// Mitsubishi GX Works2 project: BookEX6_54 Socket2   PLC: Q13UDV

// global labels: Global
VAR_GLOBAL
  bVar0 AT M5000 : BOOL;
  abArray0 AT M5010 : ARRAY [0..49] OF BOOL;
  sStr0 AT D5000 : STRING[199];
  sStr1 AT D5100 : STRING[199];
  sStr2 AT D5200 : STRING[199];
  sStr3 AT D5300 : STRING[199];
  sStr4 AT D5400 : STRING[199];
  sStr5 AT D5500 : STRING[199];
  sStr6 AT D5600 : STRING[199];
  sStr7 AT D5700 : STRING[199];
  sStr8 AT D5800 : STRING[199];
  sStr9 AT D5900 : STRING[199];
  iVar0 AT D4500 : INT;
  iVar1 AT D4501 : INT;
  iVar2 AT D4502 : INT;
  iVar3 AT D4503 : INT;
  iVar4 AT D4504 : INT;
  iVar5 AT D4505 : INT;
  iVar6 AT D4506 : INT;
  iVar7 AT D4507 : INT;
  iVar8 AT D4508 : INT;
  iVar9 AT D4509 : INT;
  dVar0 AT D4510 : DINT;
  dVar1 AT D4512 : DINT;
  dVar2 AT D4514 : DINT;
  dVar3 AT D4516 : DINT;
  dVar4 AT D4518 : DINT;
  dVar5 AT D4520 : DINT;
  dVar6 AT D4522 : DINT;
  dVar7 AT D4524 : DINT;
  dVar8 AT D4526 : DINT;
  dVar9 AT D4528 : DINT;
  wVar0 AT D4530 : WORD;
  wVar1 AT D4531 : WORD;
  wVar2 AT D4532 : WORD;
  wVar3 AT D4533 : WORD;
  wVar4 AT D4534 : WORD;
  wVar5 AT D4535 : WORD;
  wVar6 AT D4536 : WORD;
  wVar7 AT D4537 : WORD;
  wVar8 AT D4538 : WORD;
  wVar9 AT D4539 : WORD;
  dwVar0 AT D4540 : DWORD;
  dwVar1 AT D4542 : DWORD;
  dwVar2 AT D4544 : DWORD;
  dwVar3 AT D4546 : DWORD;
  dwVar4 AT D4548 : DWORD;
  dwVar5 AT D4550 : DWORD;
  dwVar6 AT D4552 : DWORD;
  dwVar7 AT D4554 : DWORD;
  dwVar8 AT D4556 : DWORD;
  dwVar9 AT D4558 : DWORD;
  fsVar0 AT D4560 : REAL;
  fsVar1 AT D4562 : REAL;
  fsVar2 AT D4564 : REAL;
  fsVar3 AT D4566 : REAL;
  fsVar4 AT D4568 : REAL;
  fsVar5 AT D4570 : REAL;
  fsVar6 AT D4572 : REAL;
  fsVar7 AT D4574 : REAL;
  fsVar8 AT D4576 : REAL;
  fsVar9 AT D4578 : REAL;
  fdVar0 AT D4580 : LREAL;
  tTime0 AT D4620 : TIME;
  tTime1 AT D4622 : TIME;
  tTime2 AT D4624 : TIME;
  tTime3 AT D4626 : TIME;
  tTime4 AT D4628 : TIME;
  tTime5 AT D4630 : TIME;
  tTime6 AT D4632 : TIME;
  tTime7 AT D4634 : TIME;
  tTime8 AT D4636 : TIME;
  tTime9 AT D4638 : TIME;
  tTime10 AT D4640 : TIME;
  bVar1 AT M5001 : BOOL;
  bVar2 AT M5002 : BOOL;
  bVar3 AT M5003 : BOOL;
  bVar4 AT M5004 : BOOL;
  bVar5 AT M5005 : BOOL;
  bVar6 AT M5006 : BOOL;
  bVar7 AT M5007 : BOOL;
  bVar8 AT M5008 : BOOL;
  bVar9 AT M5009 : BOOL;
  abArray1 AT M5060 : ARRAY [0..49] OF BOOL;
  abArray2 AT M5110 : ARRAY [0..49] OF BOOL;
  abArray3 AT M5160 : ARRAY [0..49] OF BOOL;
  abArray4 AT M5210 : ARRAY [0..49] OF BOOL;
  abArray5 AT M5260 : ARRAY [0..49] OF BOOL;
  abArray6 AT M5310 : ARRAY [0..49] OF BOOL;
  abArray7 AT M5360 : ARRAY [0..49] OF BOOL;
  abArray8 AT M5410 : ARRAY [0..49] OF BOOL;
  abArray9 AT M5460 : ARRAY [0..49] OF BOOL;
  fdVar1 AT D4584 : LREAL;
  fdVar2 AT D4588 : LREAL;
  fdVar3 AT D4592 : LREAL;
  fdVar4 AT D4596 : LREAL;
  fdVar5 AT D4600 : LREAL;
  fdVar6 AT D4604 : LREAL;
  fdVar7 AT D4608 : LREAL;
  fdVar8 AT D4612 : LREAL;
  fdVar9 AT D4616 : LREAL;
END_VAR

// global labels: QPLCSpecial
VAR_GLOBAL
  sbGetTime AT SM213 : BOOL;
  sbOn AT SM400 : BOOL;
  sbOff AT SM401 : BOOL;
  sbOn1Time AT SM402 : BOOL;
  sbOff1Time AT SM403 : BOOL;
  sb5ms AT SM409 : BOOL;
  sdSwitch AT SD200 : INT;
  sdTime03 AT SD212 : INT;
  sdTime04 AT SD213 : INT;
  sdTime02 AT SD211 : INT;
  sdTime01 AT SD210 : INT;
  sdScanTime1 AT SD521 : INT;
  sdScanTimeMin1 AT SD525 : INT;
  sdScanTimeMin AT SD524 : INT;
  sdScanTimeMax1 AT SD527 : INT;
  sdScanTimeMax AT SD526 : INT;
  sbErrInfo2 AT SM16 : BOOL;
  sbErrInfo AT SM5 : BOOL;
  sbSelfError AT SM1 : BOOL;
  sbDiagError AT SM0 : BOOL;
  sbResetErr AT SM50 : BOOL;
  sbSetTime AT SM210 : BOOL;
  sbFuse AT SM60 : BOOL;
  sbOpError AT SM56 : BOOL;
  sbPowerDown AT SM53 : BOOL;
  sbBatLow AT SM52 : BOOL;
  sbBatLowL AT SM51 : BOOL;
  sbSTOP AT SM203 : BOOL;
  sbPAUSE AT SM204 : BOOL;
  sbNsec AT SM414 : BOOL;
  sb1000ms AT SM413 : BOOL;
  sb500ms AT SM412 : BOOL;
  sbNms AT SM415 : BOOL;
  sbUserClk4 AT SM424 : BOOL;
  sbUserClk3 AT SM423 : BOOL;
  sbUserClk2 AT SM422 : BOOL;
  sbUserClk1 AT SM421 : BOOL;
  sbUserClk0 AT SM420 : BOOL;
  sdBatLowL AT SD51 : INT;
  sdPLCErrInfo AT SD4 : INT;
  sdPLCErrDate2 AT SD3 : INT;
  sdPLCErrDate1 AT SD2 : INT;
  sdPLCErrDate0 AT SD1 : INT;
  sdPLCErrCode AT SD0 : INT;
  sdFuse AT SD60 : INT;
  sdPowerDown AT SD53 : INT;
  sdBatLow AT SD52 : INT;
  sdCPUSts AT SD203 : INT;
  sdLed AT SD201 : INT;
  sdScanTime AT SD520 : INT;
  sdCntNsec AT SD414 : INT;
  sdCnt1sec AT SD412 : INT;
  sdCntScan AT SD420 : INT;
  sdCntNms AT SD415 : INT;
  sb100ms AT SM411 : BOOL;
  sb50ms AT SM410 : BOOL;
  sdSckOpenComp AT SD1282 : WORD;
  sdSckOpenReq AT SD1284 : WORD;
  sdSckDataRx AT SD1286 : WORD;
  sdSckConn AT SD1288 : WORD;
END_VAR

// global labels: Network
VAR_GLOBAL
  aSendData1 AT D100 : ARRAY [0..4] OF INT;
  aiTxData AT D4000 : ARRAY [0..99] OF INT;
  aiRxData AT D4100 : ARRAY [0..99] OF INT;
  iOpenOK AT D3900 : INT;
  iOpenERR AT D3901 : INT;
  iSendOK AT D3902 : INT;
  iSendERR AT D3903 : INT;
  iCloseOK AT D3906 : INT;
  iCloseERR AT D3907 : INT;
  iRecvOK AT D3904 : INT;
  iRecvERR AT D3905 : INT;
  aiTxData2 AT D4200 : ARRAY [0..99] OF INT;
  aiRxData2 AT D4300 : ARRAY [0..99] OF INT;
  iOpenOK2 AT D3908 : INT;
  iOpenERR2 AT D3909 : INT;
  iSendOK2 AT D3910 : INT;
  iSendERR2 AT D3911 : INT;
  iRecvOK2 AT D3912 : INT;
  iRecvERR2 AT D3913 : INT;
  iCloseOK2 AT D3914 : INT;
  iCloseERR2 AT D3915 : INT;
  iEOpenComp AT D3916 : INT;
  iEOpenReq AT D3917 : INT;
  iERecvFlag AT D3918 : INT;
  iOpenCode AT D3919 : INT;
  iSendCode AT D3920 : INT;
  iRecvCode AT D3921 : INT;
  iCloseCode AT D3922 : INT;
  iOpenCode2 AT D3923 : INT;
  iSendCode2 AT D3924 : INT;
  iRecvCode2 AT D3925 : INT;
  iCloseCode2 AT D3926 : INT;
  aRecvData1 AT D105 : ARRAY [0..4] OF INT;
  aSendData2 AT D110 : ARRAY [0..4] OF INT;
  aRecvData2 AT D115 : ARRAY [0..4] OF INT;
  aSendData3 AT D120 : ARRAY [0..4] OF INT;
  aRecvData3 AT D125 : ARRAY [0..4] OF INT;
  aRdata AT D140 : ARRAY [0..9] OF INT;
  aSLMPDataTx AT D150 : ARRAY [0..9] OF WORD;
  aSLMPDataRx AT D160 : ARRAY [0..9] OF WORD;
END_VAR
// user libraries (not included): HMI

PROGRAM Ex_READ
VAR
  Mov8INT_1 : Mov8INT;
  acRdCtrl : ARRAY [0..17] OF INT;
  abRdComp : ARRAY [0..1] OF BOOL;
  iCntRdOk : INT;
  iCntRdErr : INT;
END_VAR
(* structured ladder/FBD written out as ST: instructions are called as NAME(EN, inputs, outputs); _pN, _eN, _tN stand for wires *)
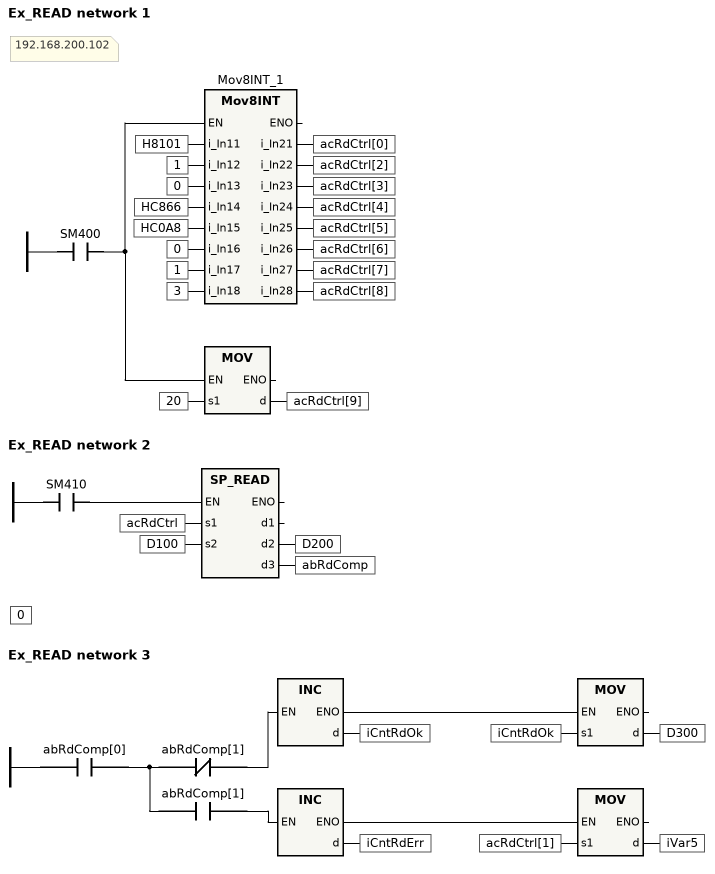
(* network 1 *)
(* 192.168.200.102 *)
Mov8INT_1(EN := SM400, i_In11 := H8101, i_In12 := 1, i_In13 := 0, i_In14 := HC866, i_In15 := HC0A8, i_In16 := 0, i_In17 := 1, i_In18 := 3, i_In21 => acRdCtrl[0], i_In22 => acRdCtrl[2], i_In23 => acRdCtrl[3], i_In24 => acRdCtrl[4], i_In25 => acRdCtrl[5], i_In26 => acRdCtrl[6], i_In27 => acRdCtrl[7], i_In28 => acRdCtrl[8]);
MOV(SM400, 20, acRdCtrl[9]);
(* network 2 *)
SP_READ(SM410, acRdCtrl, D100, _open, D200, abRdComp);
(* not connected to any output: 0 *)
(* network 3 *)
_e1 := INC(abRdComp[0] AND NOT abRdComp[1], iCntRdOk);
MOV(_e1, iCntRdOk, D300);
_e2 := INC(abRdComp[0] AND abRdComp[1], iCntRdErr);
MOV(_e2, acRdCtrl[1], iVar5);
END_PROGRAM

FUNCTION_BLOCK Word2Bit8
VAR_INPUT
  IN : WORD;
END_VAR
VAR_OUTPUT
  Bit0 : BOOL;
  Bit1 : BOOL;
  Bit2 : BOOL;
  Bit3 : BOOL;
  Bit4 : BOOL;
  Bit5 : BOOL;
  Bit6 : BOOL;
  Bit7 : BOOL;
END_VAR
 
Bit0 := WORD_TO_BOOL(IN AND 16#0001);
Bit1 := WORD_TO_BOOL(SHR(IN AND 16#0002 , 1));
Bit2 := WORD_TO_BOOL(SHR(IN AND 16#0004 , 2));
Bit3 := WORD_TO_BOOL(SHR(IN AND 16#0008 , 3));
Bit4 := WORD_TO_BOOL(SHR(IN AND 16#0010 , 4));
Bit5 := WORD_TO_BOOL(SHR(IN AND 16#0020 , 5));
Bit6 := WORD_TO_BOOL(SHR(IN AND 16#0040 , 6));
Bit7 := WORD_TO_BOOL(SHR(IN AND 16#0080 , 7));
END_FUNCTION_BLOCK

FUNCTION_BLOCK Word2Bit16
VAR_INPUT
  bEN : BOOL;
END_VAR
VAR_OUTPUT
  Bit0 : BOOL;
  Bit1 : BOOL;
  Bit2 : BOOL;
  Bit3 : BOOL;
  Bit4 : BOOL;
  Bit5 : BOOL;
  Bit6 : BOOL;
  Bit7 : BOOL;
  Bit8 : BOOL;
  Bit9 : BOOL;
  Bit10 : BOOL;
  Bit11 : BOOL;
  Bit12 : BOOL;
  Bit13 : BOOL;
  Bit14 : BOOL;
  Bit15 : BOOL;
END_VAR
VAR_INPUT
  InWord : WORD;
END_VAR
VAR_OUTPUT
  bENO : BOOL;
END_VAR
VAR
  InVal : WORD;
END_VAR
 
bENO := bEN;
InVal :=InWord;
Bit0 := (InVal AND 16#0001) = H0001;
Bit1 := (InVal AND 16#0002) = H0002;
Bit2 := (InVal AND 16#0004) = H0004;
Bit3 := (InVal AND 16#0008) = H0008;
Bit4 := (InVal AND 16#0010) = H0010;
Bit5 := (InVal AND 16#0020) = H0020;
Bit6 := (InVal AND 16#0040) = H0040;
Bit7 := (InVal AND 16#0080) = H0080;
Bit8 := (InVal AND 16#0100) = H0100;
Bit9 := (InVal AND 16#0200) = H0200;
Bit10 := (InVal AND 16#0400) = H0400;
Bit11 := (InVal AND 16#0800) = H0800;
Bit12 := (InVal AND 16#1000) = H1000;
Bit13 := (InVal AND 16#2000) = H2000;
Bit14 := (InVal AND 16#4000) = H4000;
Bit15 := (InVal AND 16#8000) = H8000;

(*
Bit0 := WORD_TO_BOOL(IN AND 16#0001);
Bit1 := WORD_TO_BOOL(SHR(IN AND 16#0002 , 1));
Bit2 := WORD_TO_BOOL(SHR(IN AND 16#0004 , 2));
Bit3 := WORD_TO_BOOL(SHR(IN AND 16#0008 , 3));
Bit4 := WORD_TO_BOOL(SHR(IN AND 16#0010 , 4));
Bit5 := WORD_TO_BOOL(SHR(IN AND 16#0020 , 5));
Bit6 := WORD_TO_BOOL(SHR(IN AND 16#0040 , 6));
Bit7 := WORD_TO_BOOL(SHR(IN AND 16#0080 , 7));
 
Bit8 := WORD_TO_BOOL(SHR(IN AND 16#0100 , 8));
Bit9 := WORD_TO_BOOL(SHR(IN AND 16#0200 , 9));
Bit10 := WORD_TO_BOOL(SHR(IN AND 16#0400 , 10));
Bit11 := WORD_TO_BOOL(SHR(IN AND 16#0800 , 11));
Bit12 := WORD_TO_BOOL(SHR(IN AND 16#1000 , 12));
Bit13 := WORD_TO_BOOL(SHR(IN AND 16#2000 , 13));
Bit14 := WORD_TO_BOOL(SHR(IN AND 16#4000 , 14));
Bit15 := WORD_TO_BOOL(SHR(IN AND 16#8000 , 15));
*)
END_FUNCTION_BLOCK

PROGRAM Ex_ECPRTCL
VAR
  bOpenReqC : BOOL;
  bOpenOkC : BOOL;
  bOpenErrC : BOOL;
  abOpenResC : ARRAY [0..1] OF BOOL;
  acOpenData : ARRAY [0..9] OF INT;
  bSendReqC : BOOL;
  bSendOkC : BOOL;
  bSendErrC : BOOL;
  abSendResC : ARRAY [0..1] OF BOOL;
  acSendDataC : ARRAY [0..1] OF INT;
  bRecvOkC : BOOL;
  bRecvErrC : BOOL;
  abRecvResC : ARRAY [0..1] OF BOOL;
  bCloseReq : BOOL;
  bCloseOkC : BOOL;
  bCloseErrC : BOOL;
  abCloseResC : ARRAY [0..1] OF BOOL;
  acCloseData : ARRAY [0..1] OF INT;
  CntSend1 : INT;
  CntSend2 : INT;
  CntRecv1 : INT;
  CntRecv2 : INT;
  Mov4INT_1 : Mov4INT;
  Mov8INT_1 : Mov8INT;
  acRdCtrl : ARRAY [0..9] OF INT;
  Mov4INT_2 : Mov4INT;
  bOpenReqE : BOOL;
  bOpenOkE : BOOL;
  bOpenErrE : BOOL;
  abOpenResE : ARRAY [0..1] OF BOOL;
  bSendErrE : BOOL;
  bSendOkE : BOOL;
  bSendReqE : BOOL;
  abSendResE : ARRAY [0..1] OF BOOL;
  abRecvResE : ARRAY [0..1] OF BOOL;
  bRecvErrE : BOOL;
  bRecvOkE : BOOL;
  abCloseResE : ARRAY [0..1] OF BOOL;
  bCloseErrE : BOOL;
  bCloseOkE : BOOL;
  acSendDataE : ARRAY [0..1] OF INT;
  acRecvDataC : ARRAY [0..1] OF INT;
  acRecvDataE : ARRAY [0..1] OF INT;
  Word2Bit8_1 : Word2Bit8;
  Word2Bit8_2 : Word2Bit8;
  Word2Bit8_3 : Word2Bit8;
  Word2Bit8_4 : Word2Bit8;
  Word2Bit8_5 : Word2Bit8;
  Word2Bit8_6 : Word2Bit8;
  ErrCodeSC : INT;
  ErrCodeSE : INT;
  Mov4INT_3 : Mov4INT;
  bChangeReqC : BOOL;
  Mov4INT_4 : Mov4INT;
  acRmodeData : ARRAY [0..3] OF INT;
  TON_1 : TON;
  CntRecvErr1 : INT;
  CntRecvErr2 : INT;
  TON_2 : TON;
  ErrCodeRC : INT;
  ErrCodeRE : INT;
  bModeReq : BOOL;
  acRdata : ARRAY [0..1] OF INT;
  bCmdReq : BOOL;
  abRes : ARRAY [0..1] OF BOOL;
  bOK : BOOL;
  bERR : BOOL;
  Mov8INT_2 : Mov8INT;
END_VAR
(* structured ladder/FBD written out as ST: instructions are called as NAME(EN, inputs, outputs); _pN, _eN, _tN stand for wires *)
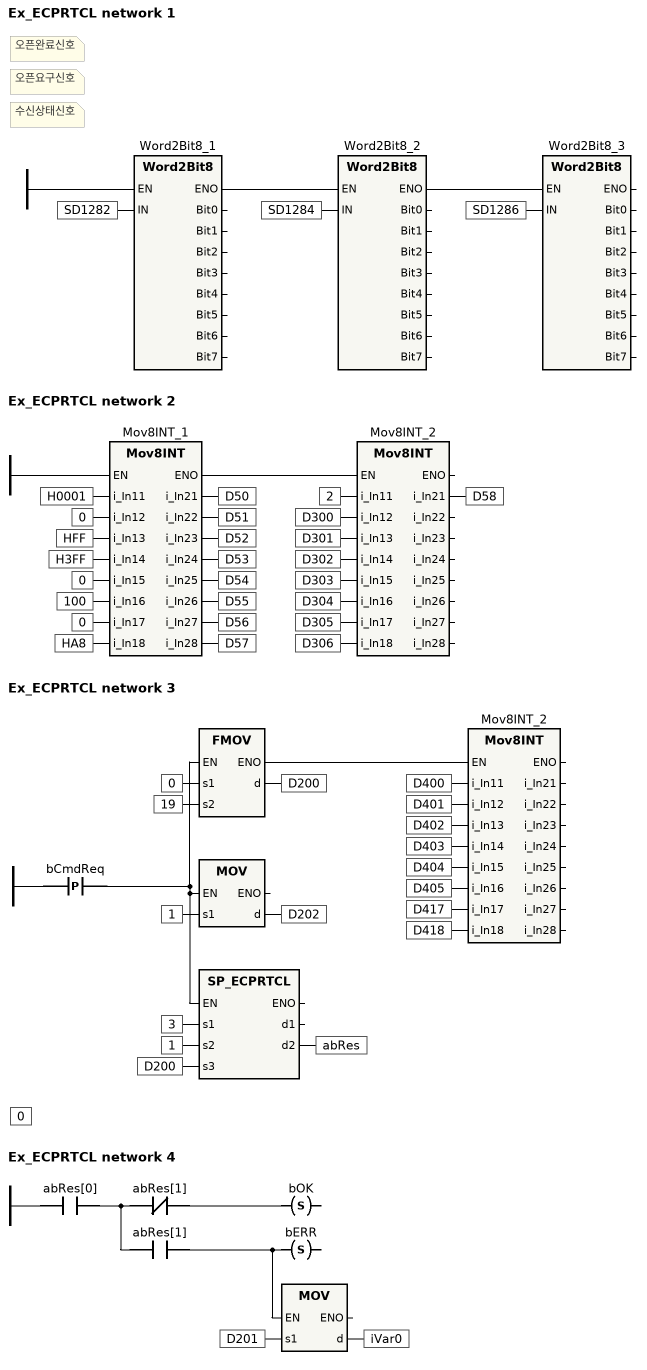
(* network 1 *)
(* 오픈완료신호 *)
(* 오픈요구신호 *)
(* 수신상태신호 *)
Word2Bit8_1(EN := TRUE, IN := SD1282);
Word2Bit8_2(EN := Word2Bit8_1.ENO, IN := SD1284);
Word2Bit8_3(EN := Word2Bit8_2.ENO, IN := SD1286);
(* network 2 *)
Mov8INT_1(EN := TRUE, i_In11 := H0001, i_In12 := 0, i_In13 := HFF, i_In14 := H3FF, i_In15 := 0, i_In16 := 100, i_In17 := 0, i_In18 := HA8, i_In21 => D50, i_In22 => D51, i_In23 => D52, i_In24 => D53, i_In25 => D54, i_In26 => D55, i_In27 => D56, i_In28 => D57);
Mov8INT_2(EN := Mov8INT_1.ENO, i_In11 := 2, i_In12 := D300, i_In13 := D301, i_In14 := D302, i_In15 := D303, i_In16 := D304, i_In17 := D305, i_In18 := D306, i_In21 => D58);
(* network 3 *)
_p1 := LDP(TRUE, bCmdReq);
_e2 := FMOV(_p1, 0, 19, D200);
Mov8INT_2(EN := _e2, i_In11 := D400, i_In12 := D401, i_In13 := D402, i_In14 := D403, i_In15 := D404, i_In16 := D405, i_In17 := D417, i_In18 := D418);
MOV(_p1, 1, D202);
SP_ECPRTCL(_p1, 3, 1, D200, _open, abRes);
(* not connected to any output: 0 *)
(* network 4 *)
SET(abRes[0] AND NOT abRes[1], bOK);
_p1 := abRes[0] AND abRes[1];
SET(_p1, bERR);
MOV(_p1, D201, iVar0);
END_PROGRAM

PROGRAM Ex_SLMPSND
VAR
  bSendReq : BOOL;
  Mov8WORD_1 : Mov8WORD;
  abSLMPRes : ARRAY [0..1] OF BOOL;
  acSLMPData : ARRAY [0..18] OF WORD;
  Mov8WORD_2 : Mov8WORD;
  Mov4WORD_1 : Mov4WORD;
  Mov8WORD_3 : Mov8WORD;
  Word2Bit16_1 : Word2Bit16;
  Word2Bit16_2 : Word2Bit16;
  Word2Bit16_3 : Word2Bit16;
  Word2Bit16_4 : Word2Bit16;
  abOpenResC : ARRAY [0..1] OF BOOL;
  abOpenResE : ARRAY [0..1] OF BOOL;
  acOpenData : ARRAY [0..9] OF INT;
  bOpenReqC : BOOL;
  bOpenOkC : BOOL;
END_VAR
(* structured ladder/FBD written out as ST: instructions are called as NAME(EN, inputs, outputs); _pN, _eN, _tN stand for wires *)
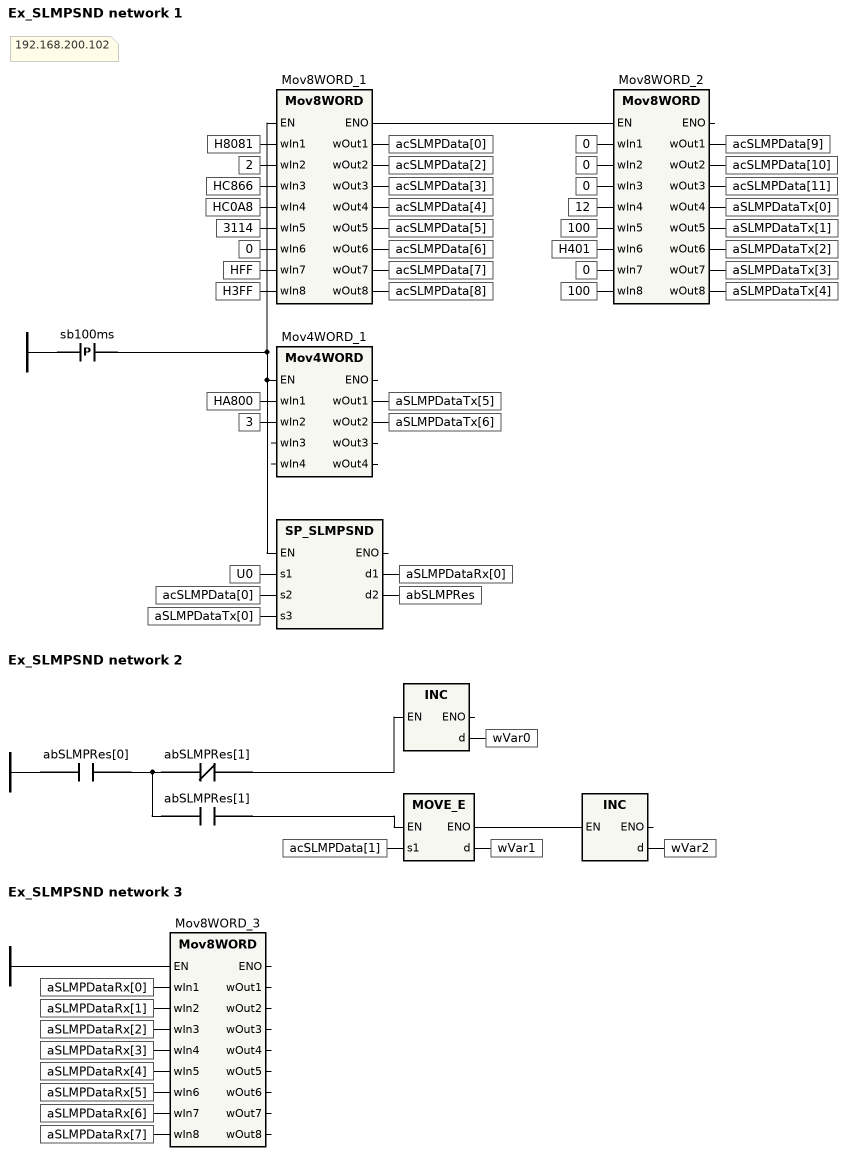
(* network 1 *)
(* 192.168.200.102 *)
_p1 := LDP(TRUE, sb100ms);
Mov8WORD_1(EN := _p1, wIn1 := H8081, wIn2 := 2, wIn3 := HC866, wIn4 := HC0A8, wIn5 := 3114, wIn6 := 0, wIn7 := HFF, wIn8 := H3FF, wOut1 => acSLMPData[0], wOut2 => acSLMPData[2], wOut3 => acSLMPData[3], wOut4 => acSLMPData[4], wOut5 => acSLMPData[5], wOut6 => acSLMPData[6], wOut7 => acSLMPData[7], wOut8 => acSLMPData[8]);
Mov8WORD_2(EN := Mov8WORD_1.ENO, wIn1 := 0, wIn2 := 0, wIn3 := 0, wIn4 := 12, wIn5 := 100, wIn6 := H401, wIn7 := 0, wIn8 := 100, wOut1 => acSLMPData[9], wOut2 => acSLMPData[10], wOut3 => acSLMPData[11], wOut4 => aSLMPDataTx[0], wOut5 => aSLMPDataTx[1], wOut6 => aSLMPDataTx[2], wOut7 => aSLMPDataTx[3], wOut8 => aSLMPDataTx[4]);
Mov4WORD_1(EN := _p1, wIn1 := HA800, wIn2 := 3, wOut1 => aSLMPDataTx[5], wOut2 => aSLMPDataTx[6]);
SP_SLMPSND(_p1, U0, acSLMPData[0], aSLMPDataTx[0], aSLMPDataRx[0], abSLMPRes);
(* network 2 *)
INC(abSLMPRes[0] AND NOT abSLMPRes[1], wVar0);
_e1 := MOVE_E(abSLMPRes[0] AND abSLMPRes[1], acSLMPData[1], wVar1);
INC(_e1, wVar2);
(* network 3 *)
Mov8WORD_3(EN := TRUE, wIn1 := aSLMPDataRx[0], wIn2 := aSLMPDataRx[1], wIn3 := aSLMPDataRx[2], wIn4 := aSLMPDataRx[3], wIn5 := aSLMPDataRx[4], wIn6 := aSLMPDataRx[5], wIn7 := aSLMPDataRx[6], wIn8 := aSLMPDataRx[7]);
END_PROGRAM

FUNCTION_BLOCK slmpDeviceRead
VAR_INPUT
  bEN : BOOL;
  dw_IPAddr : DWORD;
  i_SubCommand : INT;
  i_DeviceCode : INT;
  d_DeviceNo : DINT;
  i_DevicePoints : INT;
  i_Channel : INT;
  i_TargetPortNo : INT;
END_VAR
VAR_OUTPUT
  bENO : BOOL;
  b_OK : BOOL;
  b_ERR : BOOL;
  i_ErrCode : INT;
END_VAR
VAR
  aControlData : ARRAY [0..18] OF INT;
  aRequestData : ARRAY [0..7] OF INT;
  aResponesData : ARRAY [0..999] OF INT;
  abComp : ARRAY [0..1] OF BOOL;
  bErr1 : BOOL;
  bErr2 : BOOL;
  NoPoint : INT;
  TempDeviceCode : INT;
  bTmpErr : BOOL;
  bInputCheck : BOOL;
  bExecute : BOOL;
  bCheckEnd : BOOL;
END_VAR
VAR CONSTANT
  cRequestModuleIO : INT := H3FF;
  cResendCountMax : INT;
  cMonitorTime : INT := 1;
END_VAR
VAR
  dwTmp : DWORD;
END_VAR
VAR_OUTPUT
  i_ReadData : INT;
  i_ResendCount : INT;
  i_ErrTime : ARRAY [0..3] OF INT;
  dw_ErrIP : DWORD;
END_VAR
;
IF LDP(TRUE, bEN) AND NOT bENO THEN (*FB의 시작*)
	bENO 				:= TRUE;
	bInputCheck 	:= TRUE;
	b_OK 				:= FALSE;
	b_ERR 				:= FALSE;
	i_ErrCode 		:= 0;
	bTmpErr 			:= FALSE;
END_IF;

IF NOT bEN THEN (*FB의 종료*)
	b_OK 				:= FALSE;
	b_ERR 				:= FALSE;
	i_ErrCode 		:= 0;
 	bTmpErr 			:= FALSE;
	bENO 				:= FALSE;
	bInputCheck 	:= FALSE;
	bCheckEnd 	:= FALSE;
	bExecute 			:= FALSE;
END_IF;

IF LDP(TRUE, bInputCheck) THEN
	IF i_SubCommand < 0 OR i_SubCommand > 1 										THEN i_ErrCode := 11; END_IF;
	IF i_DeviceCode < 0 OR i_DeviceCode > WORD_TO_INT(HFF) 	THEN i_ErrCode := 12; END_IF;
	IF d_DeviceNo < 0 OR d_DeviceNo > DWORD_TO_DINT(HFFFFFF) 	THEN i_ErrCode := 13; END_IF;
	IF i_DevicePoints < 1 OR i_DevicePoints > 960 									THEN i_ErrCode := 14; END_IF;
	IF i_Channel < 1 OR i_Channel > 9 																THEN i_ErrCode := 15; END_IF;
	IF i_TargetPortNo = 0 OR i_TargetPortNo = HFFFF 							THEN i_ErrCode := 16; END_IF;
	IF i_ErrCode <> 0 THEN 		
		bTmpErr := TRUE;
	END_IF;	  
	bCheckEnd := bTmpErr = 0;
END_IF;			
		
IF LDP(TRUE, bCheckEnd) THEN
	FMOV(TRUE, 0, 19, aControlData[0]);		
	aControlData[0] 	:= H8081;
	aControlData[2] 	:= i_Channel;
	aControlData[3] 	:= DWORD_TO_INT(dw_IPAddr AND H0000FFFF);
	aControlData[4] 	:= DWORD_TO_INT(SHR(dw_IPAddr,16) AND H0000FFFF);
	aControlData[5] 	:= i_TargetPortNo;	
	aControlData[6] 	:= 0;	
	aControlData[7] 	:= HFF;	
	aControlData[8] 	:= cRequestModuleIO;	
	aControlData[9] 	:= 0;	
	aControlData[10] 	:= cResendCountMax;
	aControlData[11] 	:= cMonitorTime;

	aRequestData[0] := 12;
	aRequestData[1] := 2;
	aRequestData[2] := H401;
	aRequestData[3] := i_SubCommand;
	dwTmp := DINT_TO_DWORD( d_DeviceNo);
	aRequestData[4] := DWORD_TO_INT(dwTmp AND H0000FFFF);
	aRequestData[5] := DWORD_TO_INT(SHR(dwTmp,16) AND H0000FFFF);
	IF i_SubCommand = 0 THEN 
		NoPoint := i_DevicePoints; 
	ELSIF i_SubCommand = 1 THEN 
		NoPoint := i_DevicePoints+3; 
		NoPoint := i_DevicePoints / 4; 
	END_IF;
	TempDeviceCode := i_DeviceCode;
	SFL(TRUE, 8, TempDeviceCode);
	WOR(TRUE, TempDeviceCode, aRequestData[5], aRequestData[5]);
	aRequestData[6] := NoPoint;
	bExecute := TRUE;
END_IF;
			
SP_SLMPSND( bExecute, "U0", aControlData[0], aRequestData[0], aResponesData[0], abComp);  (*상승에지에서 실행*)
IF abComp[0] THEN	(*실행 완료 *)
	i_ErrCode 			:= aControlData[1];
	i_ResendCount 	:= aControlData[10];
	BMOV(TRUE, aControlData[13], 4, i_ErrTime[0]); 
	dw_ErrIP := INT_TO_DWORD(aControlData[17]) OR SHL(INT_TO_DWORD( aControlData[18]),16);
	bExecute 				:= FALSE;
	IF abComp[1] THEN
		bErr2 					:= TRUE;		(* 이상완료*)
	ELSE								(* 정상완료*)
		IF aResponesData[1] = 0 THEN
			b_OK 			:=TRUE;
		 	BMOV( TRUE, aResponesData[2], NoPoint, i_ReadData );
		ELSE
			i_ErrCode 	:= aResponesData[1];		(*에러코드*)
			bErr1 				:= TRUE; 
		END_IF;
	END_IF;
END_IF;

IF bTmpErr OR bErr1 OR bErr2 THEN
 	b_ERR 		:= TRUE;
 	bErr1 			:= FALSE;
  	bErr2 			:= FALSE;
END_IF;
END_FUNCTION_BLOCK

PROGRAM Ex_OtherUDV
VAR
  Mov8INT_1 : Mov8INT;
  Mov8INT_2 : Mov8INT;
END_VAR
(* structured ladder/FBD written out as ST: instructions are called as NAME(EN, inputs, outputs); _pN, _eN, _tN stand for wires *)
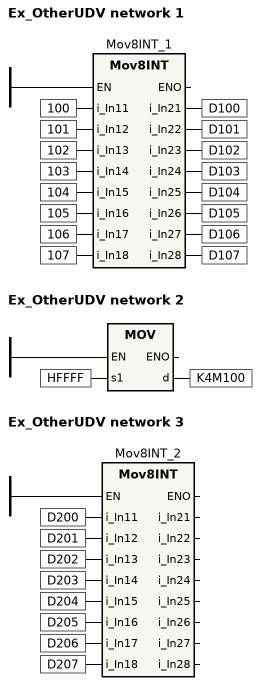
(* network 1 *)
Mov8INT_1(EN := TRUE, i_In11 := 100, i_In12 := 101, i_In13 := 102, i_In14 := 103, i_In15 := 104, i_In16 := 105, i_In17 := 106, i_In18 := 107, i_In21 => D100, i_In22 => D101, i_In23 => D102, i_In24 => D103, i_In25 => D104, i_In26 => D105, i_In27 => D106, i_In28 => D107);
(* network 2 *)
MOV(TRUE, HFFFF, K4M100);
(* network 3 *)
Mov8INT_2(EN := TRUE, i_In11 := D200, i_In12 := D201, i_In13 := D202, i_In14 := D203, i_In15 := D204, i_In16 := D205, i_In17 := D206, i_In18 := D207);
END_PROGRAM

PROGRAM Ex_DeviceRead
VAR
  slmpDeviceRead_1 : slmpDeviceRead;
  bRun : BOOL;
  bOK : BOOL;
  bERR : BOOL;
  ErrCode : INT;
  bSetErr : BOOL;
  bExeReq : BOOL;
  ResendCount : INT;
  ErrTime : ARRAY [0..3] OF INT;
  ErrIP : DWORD;
  Mov4INT_1 : Mov4INT;
  Mov4INT_2 : Mov4INT;
END_VAR
(* structured ladder/FBD written out as ST: instructions are called as NAME(EN, inputs, outputs); _pN, _eN, _tN stand for wires *)
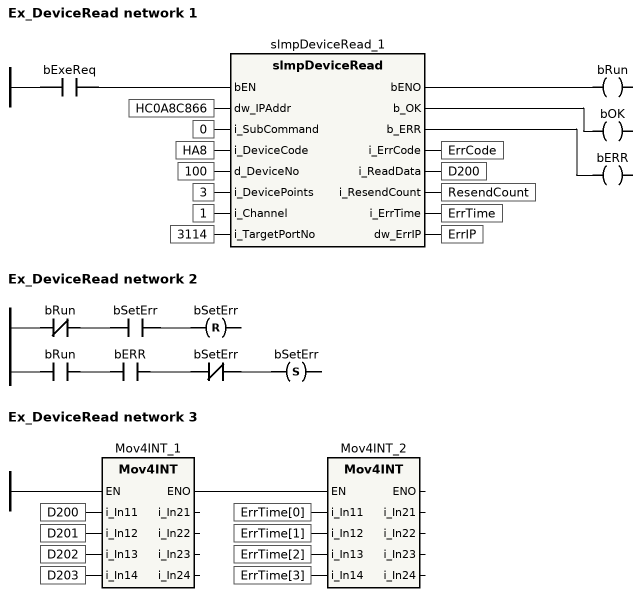
(* network 1 *)
slmpDeviceRead_1(bEN := bExeReq, dw_IPAddr := HC0A8C866, i_SubCommand := 0, i_DeviceCode := HA8, d_DeviceNo := 100, i_DevicePoints := 3, i_Channel := 1, i_TargetPortNo := 3114, i_ErrCode => ErrCode, i_ReadData => D200, i_ResendCount => ResendCount, i_ErrTime => ErrTime, dw_ErrIP => ErrIP);
bRun := slmpDeviceRead_1.bENO;
bOK := slmpDeviceRead_1.b_OK;
bERR := slmpDeviceRead_1.b_ERR;
(* network 2 *)
RST(NOT bRun AND bSetErr, bSetErr);
SET(bRun AND bERR AND NOT bSetErr, bSetErr);
(* network 3 *)
Mov4INT_1(EN := TRUE, i_In11 := D200, i_In12 := D201, i_In13 := D202, i_In14 := D203);
Mov4INT_2(EN := Mov4INT_1.ENO, i_In11 := ErrTime[0], i_In12 := ErrTime[1], i_In13 := ErrTime[2], i_In14 := ErrTime[3]);
END_PROGRAM

FUNCTION_BLOCK slmpDeviceWrite
VAR_INPUT
  bEN : BOOL;
  dw_IPAddr : DWORD;
  i_SubCommand : INT;
  i_DeviceCode : INT;
  d_DeviceNo : DINT;
  i_DevicePoints : INT;
  i_Channel : INT;
  i_TargetPortNo : INT;
END_VAR
VAR_OUTPUT
  bENO : BOOL;
  b_OK : BOOL;
  b_ERR : BOOL;
  i_ErrCode : INT;
END_VAR
VAR
  aControlData : ARRAY [0..18] OF INT;
  aRequestData : ARRAY [0..999] OF INT;
  aResponesData : ARRAY [0..6] OF INT;
  abComp : ARRAY [0..1] OF BOOL;
  NoWritePoint : INT;
  TempDeviceCode : INT;
  bTmpErr : BOOL;
  bInputCheck : BOOL;
  bExecute : BOOL;
  bCheckEnd : BOOL;
END_VAR
VAR CONSTANT
  cRequestModuleIO : INT := H3FF;
  cResendCountMax : INT;
  cMonitorTime : INT := 1;
END_VAR
VAR
  dwTmp : DWORD;
END_VAR
VAR_INPUT
  i_WriteData : INT;
END_VAR
VAR
  NoWriteLength : INT;
END_VAR
VAR_OUTPUT
  i_ResendCount : INT;
  i_ErrTime : ARRAY [0..3] OF INT;
  dw_ErrIP : DWORD;
END_VAR
VAR
  bErr1 : BOOL;
  bErr2 : BOOL;
END_VAR
;
IF LDP(TRUE, bEN) AND NOT bENO THEN (*FB의 시작*)
	bENO 				:= TRUE;
	bInputCheck 	:= TRUE;
	b_OK 				:= FALSE;
	b_ERR 				:= FALSE;
	i_ErrCode 		:= 0;
	bTmpErr 			:= FALSE;
END_IF;

IF NOT bEN THEN (*FB의 종료*)
	b_OK 				:= FALSE;
	b_ERR 				:= FALSE;
	i_ErrCode 		:= 0;
 	bTmpErr 			:= FALSE;
	bENO 				:= FALSE;
	bInputCheck 	:= FALSE;
	bCheckEnd 	:= FALSE;
	bExecute 			:= FALSE;
END_IF;

IF LDP(TRUE, bInputCheck) THEN
	IF i_SubCommand < 0 OR i_SubCommand > 1 										THEN i_ErrCode := 11; END_IF;
	IF i_DeviceCode < 0 OR i_DeviceCode > WORD_TO_INT(HFF) 	THEN i_ErrCode := 12; END_IF;
	IF d_DeviceNo < 0 OR d_DeviceNo > DWORD_TO_DINT(HFFFFFF) 	THEN i_ErrCode := 13; END_IF;
	IF i_DevicePoints < 1 OR i_DevicePoints > 960 									THEN i_ErrCode := 14; END_IF;
	IF i_Channel < 1 OR i_Channel > 9 																THEN i_ErrCode := 15; END_IF;
	IF i_TargetPortNo = 0 OR i_TargetPortNo = HFFFF 							THEN i_ErrCode := 16; END_IF;
	IF i_ErrCode <> 0 THEN 		
		bTmpErr := TRUE;
	END_IF;	  
	bCheckEnd := bTmpErr = 0;
END_IF;			
		
IF LDP(TRUE, bCheckEnd) THEN
	FMOV(TRUE, 0, 19, aControlData[0]);		
	aControlData[0] 	:= H8081;
	aControlData[2] 	:= i_Channel;
	aControlData[3] 	:= DWORD_TO_INT(dw_IPAddr AND H0000FFFF);
	aControlData[4] 	:= DWORD_TO_INT(SHR(dw_IPAddr,16) AND H0000FFFF);
	aControlData[5] 	:= i_TargetPortNo;	
	aControlData[6] 	:= 0;	
	aControlData[7] 	:= HFF;	
	aControlData[8] 	:= cRequestModuleIO;	
	aControlData[9] 	:= 0;	
	aControlData[10] 	:= cResendCountMax;
	aControlData[11] 	:= cMonitorTime;

	aRequestData[0] := 12;
	aRequestData[1] := 2;
	aRequestData[2] := H1401;
	aRequestData[3] := i_SubCommand;
	dwTmp := DINT_TO_DWORD( d_DeviceNo);
	aRequestData[4] := DWORD_TO_INT(dwTmp AND H0000FFFF);
	aRequestData[5] := DWORD_TO_INT(SHR(dwTmp,16) AND H0000FFFF);
	IF i_SubCommand = 0 THEN 
		NoWritePoint := i_DevicePoints; 
		NoWriteLength := NoWritePoint * 2;
	ELSIF i_SubCommand = 1 THEN 
		NoWritePoint := i_DevicePoints+3; 
		NoWritePoint := NoWritePoint / 4;
		NoWriteLength := i_DevicePoints + 1; 
		NoWriteLength := NoWriteLength / 2; 
	END_IF;
	aRequestData[0] := aRequestData[0] + NoWriteLength;
	TempDeviceCode := i_DeviceCode;
	SFL(TRUE, 8, TempDeviceCode);
	WOR(TRUE, TempDeviceCode, aRequestData[5], aRequestData[5]);
	aRequestData[6] := i_DevicePoints;
	BMOV(TRUE, i_WriteData, NoWritePoint, aRequestData[7]); 
	bExecute := TRUE;
END_IF;
			
SP_SLMPSND( bExecute, "U0", aControlData[0], aRequestData[0], aResponesData[0], abComp);  (*상승에지에서 실행*)
IF abComp[0] THEN	(*실행 완료 *)
	i_ErrCode 			:= aControlData[1];
	i_ResendCount 	:= aControlData[10];
	BMOV(TRUE, aControlData[13], 4, i_ErrTime[0]); 
	dw_ErrIP := INT_TO_DWORD(aControlData[17]) OR SHL(INT_TO_DWORD( aControlData[18]),16);
	bExecute 				:= FALSE;
	IF abComp[1] THEN
		bErr2 					:= TRUE;		(* 이상완료*)
	ELSE								(* 정상완료*)
		IF aResponesData[1] = 0 THEN
			b_OK 			:=TRUE;
		ELSE
			i_ErrCode 	:= aResponesData[1];		(*에러코드*)
			bErr1 				:= TRUE; 
		END_IF;
	END_IF;
END_IF;

IF bTmpErr OR bErr1 OR bErr2 THEN
 	b_ERR 		:= TRUE;
 	bErr1 			:= FALSE;
  	bErr2 			:= FALSE;
END_IF;
END_FUNCTION_BLOCK

FUNCTION_BLOCK slmpRemoteReset
VAR_INPUT
  bEN : BOOL;
  dw_IPAddr : DWORD;
  i_Channel : INT;
  i_TargetPortNo : INT;
END_VAR
VAR_OUTPUT
  bENO : BOOL;
  b_OK : BOOL;
  b_ERR : BOOL;
  i_ErrCode : INT;
END_VAR
VAR
  aControlData : ARRAY [0..18] OF INT;
  aRequestData : ARRAY [0..4] OF INT;
  aResponesData : ARRAY [0..6] OF INT;
  abComp : ARRAY [0..1] OF BOOL;
  NoPoint : INT;
  bInputCheck : BOOL;
  bExecute : BOOL;
  bCheckEnd : BOOL;
END_VAR
VAR CONSTANT
  cRequestModuleIO : INT := H3FF;
  cResendCountMax : INT;
  cMonitorTime : INT := 1;
END_VAR
VAR_OUTPUT
  i_ResendCount : INT;
  i_ErrTime : ARRAY [0..3] OF INT;
  dw_ErrIP : DWORD;
END_VAR
;
IF LDP(TRUE, bEN) AND NOT bENO THEN (*FB의 시작*)
	bENO 				:= TRUE;
	bInputCheck 	:= TRUE;
	bExecute 			:= FALSE;
END_IF;

IF NOT bEN THEN (*FB의 종료*)
	b_OK 				:= FALSE;
	b_ERR 				:= FALSE;
	i_ErrCode 		:= 0;
	bENO 				:= FALSE;
	bInputCheck 	:= FALSE;
	bCheckEnd 	:= FALSE;
	bExecute 			:= FALSE;
END_IF;

IF LDP(TRUE, bInputCheck) THEN
	IF i_Channel < 1 OR i_Channel > 9 																THEN i_ErrCode := 15; END_IF;
	IF i_TargetPortNo = 0 OR i_TargetPortNo = HFFFF 							THEN i_ErrCode := 16; END_IF;
	bCheckEnd := i_ErrCode = 0;
END_IF;			
		
IF LDP(TRUE, bCheckEnd) THEN
	FMOV(TRUE, 0, 19, aControlData[0]);		
	aControlData[0] 	:= H8080;
	aControlData[2] 	:= i_Channel;
	aControlData[3] 	:= DWORD_TO_INT(dw_IPAddr AND H0000FFFF);
	aControlData[4] 	:= DWORD_TO_INT(SHR(dw_IPAddr,16) AND H0000FFFF);
	aControlData[5] 	:= i_TargetPortNo;	
	aControlData[6] 	:= 0;	
	aControlData[7] 	:= HFF;	
	aControlData[8] 	:= cRequestModuleIO;	
	aControlData[9] 	:= 0;	
	aControlData[10] 	:= cResendCountMax;
	aControlData[11] 	:= cMonitorTime;

	aRequestData[0] := 8;
	aRequestData[1] := 2;
	aRequestData[2] := H1006;
	aRequestData[3] := 0;
	aRequestData[4] := 1;
	bExecute := TRUE;
	bCheckEnd := FALSE;
END_IF;
			
SP_SLMPSND( bExecute, "U0", aControlData[0], aRequestData[0], aResponesData[0], abComp);  (*상승에지에서 실행*)
IF abComp[0] THEN	(*실행 완료 *)
	bExecute 				:= FALSE;
	IF abComp[1] THEN	(* 이상완료*)
		i_ErrCode 			:= aControlData[1];
		i_ResendCount 	:= aControlData[10];
		BMOV(TRUE, aControlData[13], 4, i_ErrTime[0]); 
		dw_ErrIP := INT_TO_DWORD(aControlData[17]) OR SHL(INT_TO_DWORD( aControlData[18]),16);
	ELSE								(* 정상완료*)
		b_OK 			:=TRUE;
	END_IF;
END_IF;

IF i_ErrCode <> 0 THEN
 	b_ERR 		:= TRUE;
END_IF;
END_FUNCTION_BLOCK

PROGRAM Ex_DeviceWrite
VAR
  slmpDeviceRead_1 : slmpDeviceRead;
  bRun : BOOL;
  bOK : BOOL;
  bERR : BOOL;
  ErrCode : INT;
  bSetErr : BOOL;
  bExeReq : BOOL;
  ResendCount : INT;
  ErrTime : ARRAY [0..3] OF INT;
  ErrIP : DWORD;
  Mov4INT_1 : Mov4INT;
  Mov4INT_2 : Mov4INT;
  slmpDeviceWrite_1 : slmpDeviceWrite;
  Mov4INT_3 : Mov4INT;
  bExeReq2 : BOOL;
END_VAR
(* structured ladder/FBD written out as ST: instructions are called as NAME(EN, inputs, outputs); _pN, _eN, _tN stand for wires *)
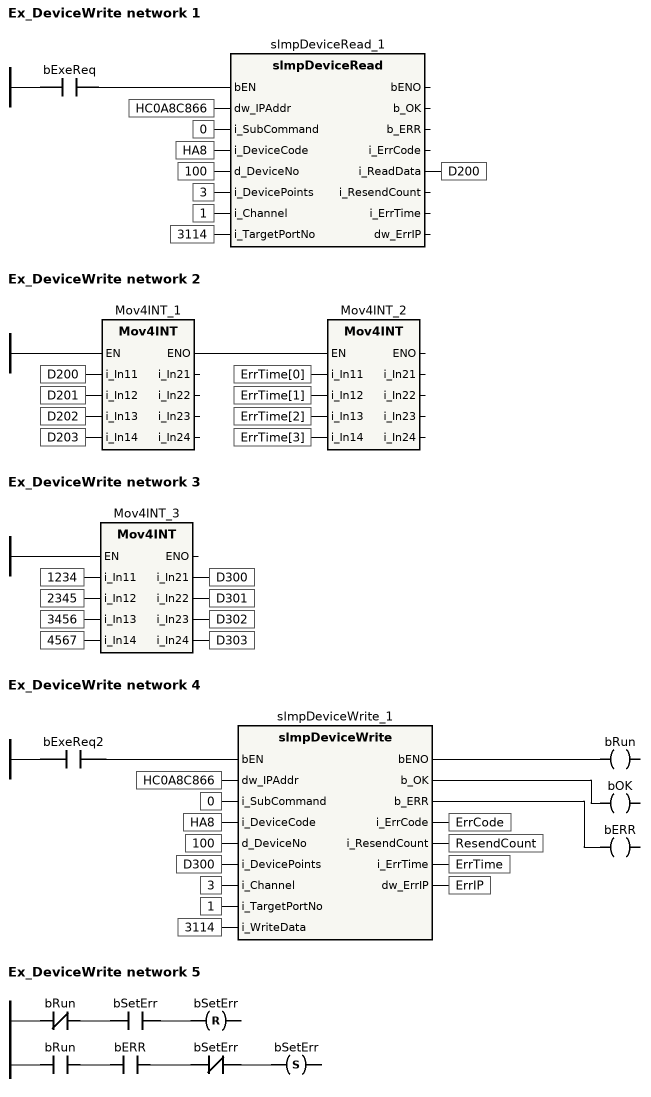
(* network 1 *)
slmpDeviceRead_1(bEN := bExeReq, dw_IPAddr := HC0A8C866, i_SubCommand := 0, i_DeviceCode := HA8, d_DeviceNo := 100, i_DevicePoints := 3, i_Channel := 1, i_TargetPortNo := 3114, i_ReadData => D200);
(* network 2 *)
Mov4INT_1(EN := TRUE, i_In11 := D200, i_In12 := D201, i_In13 := D202, i_In14 := D203);
Mov4INT_2(EN := Mov4INT_1.ENO, i_In11 := ErrTime[0], i_In12 := ErrTime[1], i_In13 := ErrTime[2], i_In14 := ErrTime[3]);
(* network 3 *)
Mov4INT_3(EN := TRUE, i_In11 := 1234, i_In12 := 2345, i_In13 := 3456, i_In14 := 4567, i_In21 => D300, i_In22 => D301, i_In23 => D302, i_In24 => D303);
(* network 4 *)
slmpDeviceWrite_1(bEN := bExeReq2, dw_IPAddr := HC0A8C866, i_SubCommand := 0, i_DeviceCode := HA8, d_DeviceNo := 100, i_DevicePoints := D300, i_Channel := 3, i_TargetPortNo := 1, i_WriteData := 3114, i_ErrCode => ErrCode, i_ResendCount => ResendCount, i_ErrTime => ErrTime, dw_ErrIP => ErrIP);
bRun := slmpDeviceWrite_1.bENO;
bOK := slmpDeviceWrite_1.b_OK;
bERR := slmpDeviceWrite_1.b_ERR;
(* network 5 *)
RST(NOT bRun AND bSetErr, bSetErr);
SET(bRun AND bERR AND NOT bSetErr, bSetErr);
END_PROGRAM

PROGRAM Ex_RemoteReset
VAR
  bRun : BOOL;
  bOK : BOOL;
  bERR : BOOL;
  ErrCode : INT;
  bSetErr : BOOL;
  bExeReq : BOOL;
  ResendCount : INT;
  ErrTime : ARRAY [0..3] OF INT;
  ErrIP : DWORD;
  Mov4INT_1 : Mov4INT;
  Mov4INT_2 : Mov4INT;
  slmpRemoteReset_1 : slmpRemoteReset;
END_VAR
(* structured ladder/FBD written out as ST: instructions are called as NAME(EN, inputs, outputs); _pN, _eN, _tN stand for wires *)
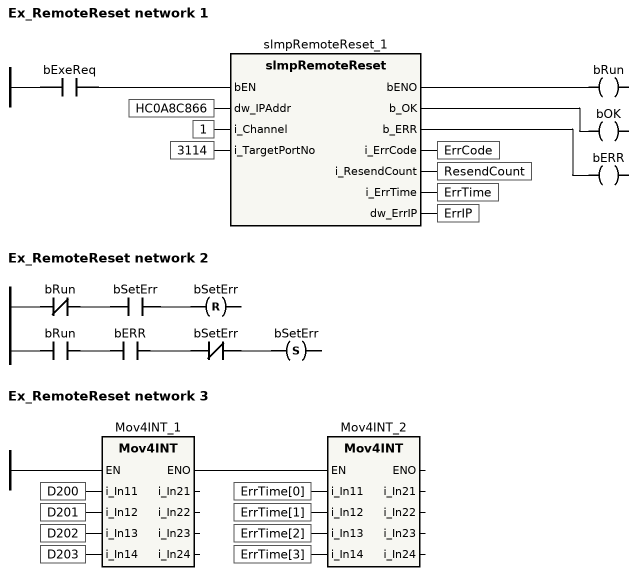
(* network 1 *)
slmpRemoteReset_1(bEN := bExeReq, dw_IPAddr := HC0A8C866, i_Channel := 1, i_TargetPortNo := 3114, i_ErrCode => ErrCode, i_ResendCount => ResendCount, i_ErrTime => ErrTime, dw_ErrIP => ErrIP);
bRun := slmpRemoteReset_1.bENO;
bOK := slmpRemoteReset_1.b_OK;
bERR := slmpRemoteReset_1.b_ERR;
(* network 2 *)
RST(NOT bRun AND bSetErr, bSetErr);
SET(bRun AND bERR AND NOT bSetErr, bSetErr);
(* network 3 *)
Mov4INT_1(EN := TRUE, i_In11 := D200, i_In12 := D201, i_In13 := D202, i_In14 := D203);
Mov4INT_2(EN := Mov4INT_1.ENO, i_In11 := ErrTime[0], i_In12 := ErrTime[1], i_In13 := ErrTime[2], i_In14 := ErrTime[3]);
END_PROGRAM

PROGRAM Ex_WRITE
VAR
  Mov8INT_1 : Mov8INT;
  acCtrlData : ARRAY [0..17] OF INT;
  iCntWrOk : INT;
  iCntWrErr : INT;
  abRes : ARRAY [0..1] OF BOOL;
  Mov8INT_2 : Mov8INT;
END_VAR
(* structured ladder/FBD written out as ST: instructions are called as NAME(EN, inputs, outputs); _pN, _eN, _tN stand for wires *)
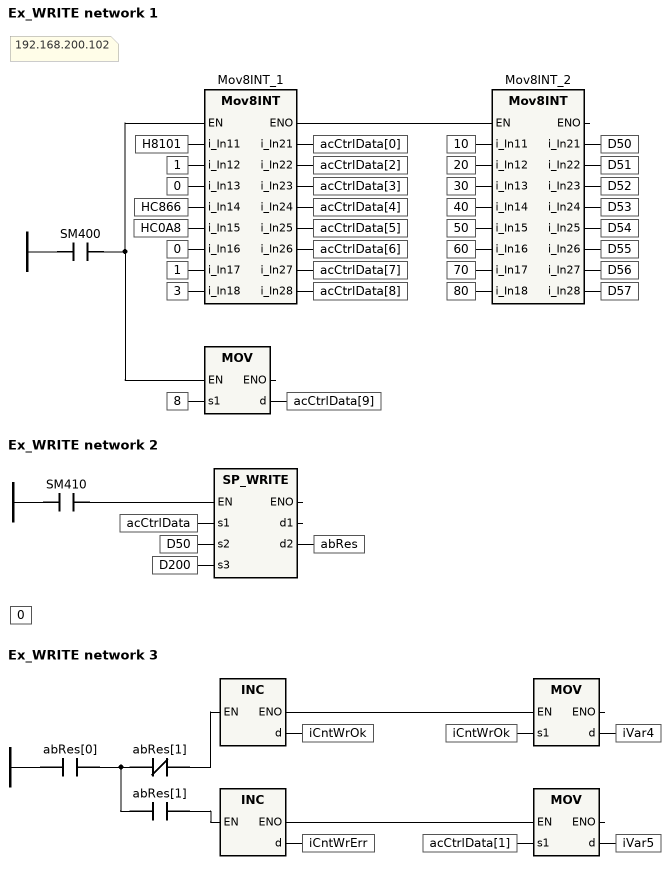
(* network 1 *)
(* 192.168.200.102 *)
Mov8INT_1(EN := SM400, i_In11 := H8101, i_In12 := 1, i_In13 := 0, i_In14 := HC866, i_In15 := HC0A8, i_In16 := 0, i_In17 := 1, i_In18 := 3, i_In21 => acCtrlData[0], i_In22 => acCtrlData[2], i_In23 => acCtrlData[3], i_In24 => acCtrlData[4], i_In25 => acCtrlData[5], i_In26 => acCtrlData[6], i_In27 => acCtrlData[7], i_In28 => acCtrlData[8]);
Mov8INT_2(EN := Mov8INT_1.ENO, i_In11 := 10, i_In12 := 20, i_In13 := 30, i_In14 := 40, i_In15 := 50, i_In16 := 60, i_In17 := 70, i_In18 := 80, i_In21 => D50, i_In22 => D51, i_In23 => D52, i_In24 => D53, i_In25 => D54, i_In26 => D55, i_In27 => D56, i_In28 => D57);
MOV(SM400, 8, acCtrlData[9]);
(* network 2 *)
SP_WRITE(SM410, acCtrlData, D50, D200, _open, abRes);
(* not connected to any output: 0 *)
(* network 3 *)
_e1 := INC(abRes[0] AND NOT abRes[1], iCntWrOk);
MOV(_e1, iCntWrOk, iVar4);
_e2 := INC(abRes[0] AND abRes[1], iCntWrErr);
MOV(_e2, acCtrlData[1], iVar5);
END_PROGRAM
